// TIA Portal V19 export
FUNCTION "DoorSignals" : Void   // FC79, LAD
// stored: Access Published, SetENOAutomatically false
   VAR_INPUT
      Door : "udt_DoorSts";
      TwoHandEnable : Bool;
   END_VAR
   VAR_OUTPUT
      LampEntry : Bool;   // Entry request lamp
      LampRst : Bool;   // Reset door lamp
   END_VAR
BEGIN

REGION Network 1: Lamps Door / Lamps Door 01 - Decoiler Front
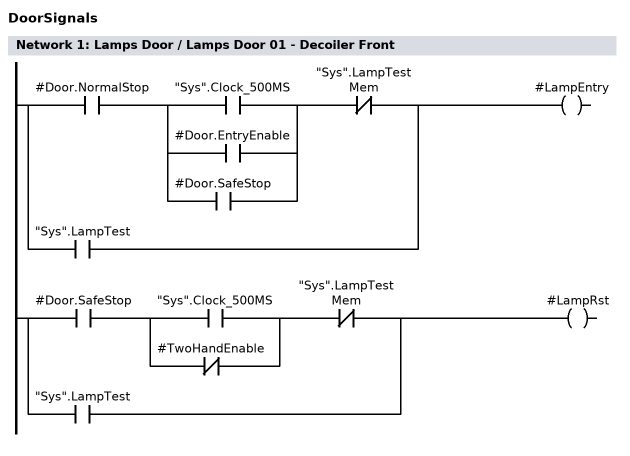
   RUNG wire#powerrail
      Contact( #Door.NormalStop )
      wire#w1
      Contact( "Sys".Clock_500MS )
      wire#w2
      I_Contact( "Sys".LampTestMem )
      wire#w3
      Coil( #LampEntry )
   END_RUNG
   RUNG wire#w1
      Contact( #Door.EntryEnable )
   END_RUNG wire#w2
   RUNG wire#w1
      Contact( #Door.SafeStop )
   END_RUNG wire#w2
   RUNG wire#powerrail
      Contact( "Sys".LampTest )
   END_RUNG wire#w3
   RUNG wire#powerrail
      Contact( #Door.SafeStop )
      wire#w4
      Contact( "Sys".Clock_500MS )
      wire#w5
      I_Contact( "Sys".LampTestMem )
      wire#w6
      Coil( #LampRst )
   END_RUNG
   RUNG wire#w4
      I_Contact( #TwoHandEnable )
   END_RUNG wire#w5
   RUNG wire#powerrail
      Contact( "Sys".LampTest )
   END_RUNG wire#w6
   // the same network as SCL:
   #LampEntry := (#Door.NormalStop AND ("Sys".Clock_500MS OR #Door.EntryEnable OR #Door.SafeStop) AND NOT "Sys".LampTestMem) OR "Sys".LampTest;
   #LampRst := (#Door.SafeStop AND ("Sys".Clock_500MS OR NOT #TwoHandEnable) AND NOT "Sys".LampTestMem) OR "Sys".LampTest;
END_REGION
END_FUNCTION
